FUNCTION_BLOCK FB_EventLogger EXTENDS FB_Cycle IMPLEMENTS I_Logger
VAR_INPUT
END_VAR
VAR_OUTPUT
END_VAR
VAR
	nLength:		INT;
	aEvent:						ARRAY [0..99] OF ST_Event;
END_VAR

METHOD PUBLIC M_Cycle
VAR_INPUT
END_VAR
VAR
	nIndex: 	DINT;
END_VAR
//nIndex:= 0;
//WHILE nIndex < nLength DO
//	IF aEvent[nIndex].Active THEN
//		CASE aEvent[nIndex].EventType OF
//			E_Event.Error:;
//			ELSE
//				aEvent[nIndex].Active:= FALSE;		
//		END_CASE		
	
	
//	ELSE
//		Tc2_System.MEMSet(ADR(aEvent[nIndex]), 0, SIZEOF(ST_Event));
//	END_IF
//	nIndex := nIndex + 1;
//END_WHILE
END_METHOD

METHOD M_Find : DINT
VAR_INPUT
	stEvent	: 		ST_Event;
END_VAR
VAR
	nIndex: 	DINT;
END_VAR
// Object already in List
M_Find := -1;
nIndex:= 0;
WHILE nIndex < nLength DO
    IF (aEvent[nIndex].Source = stEvent.Source) 
		AND_THEN (aEvent[nIndex].EventType = stEvent.EventType) 
		AND_THEN (aEvent[nIndex].Message = stEvent.Message) THEN
			M_Find := nIndex;
			RETURN;
    END_IF
	nIndex := nIndex + 1;
END_WHILE
END_METHOD

METHOD M_Log
VAR_INPUT
	stEvent	: 		ST_Event;
END_VAR

VAR
	nIndex: DINT;
END_VAR
IF M_Find(stEvent) = -1 THEN
	aEvent[nLength]:= stEvent;
	nLength:= nLength + 1;
END_IF
END_METHOD

METHOD PUBLIC M_Reset
VAR_INPUT
END_VAR
VAR
	nIndex: 	DINT;
END_VAR
//nIndex:= 0;
//WHILE nIndex < nLength DO
//	IF 	aEvent[nIndex].Active THEN
//		aEvent[nIndex].Active:= FALSE;
//	END_IF
//	nIndex := nIndex + 1;
//END_WHILE
nLength:= 0;
Tc2_System.MEMSET(ADR(aEvent), 0, SIZEOF(nLength));
END_METHOD

END_FUNCTION_BLOCK

(* stored: Version 1.1.0.1
   POU FB_EventLogger: Id {0de6697e-1d44-0296-1f4b-99ef100b1e6c}, SpecialFunc None
   Method M_Cycle: Id {2604dc42-e042-0a11-3bad-be2964c0960e}
   Method M_Find: Id {c7fd1c8c-04f0-0d78-3ad7-f0e13fc431d5}
   Method M_Log: Id {8d3f3c1a-c9ab-0738-1814-9d0b65b7b611}
   Method M_Reset: Id {e98b1693-4b94-09ac-0147-67fd83f8819f} *)
